{attribute 'GeneratedUsingTerminal: AT2042-0250-0024'}
{attribute addProperty BoxType "AT2042-0250-0024"}
{attribute addProperty Id "A_0098_AT2025_5250_0019_AT2025_5250AT2025_33A3DF1B80"}
{attribute addProperty CRC "455135025"}
{attribute addProperty Size "80"}
TYPE A_0046_AT2042_0250_0024_1B20CF31 EXTENDS AT2042_2EA6C9BF :
STRUCT
	{attribute addProperty Name "A_0098_AT2025_5250_0019_AT2025_5250"}
	A_0098_AT2025_5250_0019_AT2025_5250 : AT2025_33A3DF1B;
END_STRUCT
END_TYPE

(* stored: Version 1.2.0.0, ProductVersion 3.1.4024.9
   DUT A_0046_AT2042_0250_0024_1B20CF31: Id {26f9a2d5-ceab-4da9-abbc-6194770403d5} *)
